INTERFACE I_PersistentEventStorage

METHOD StoreEvent
VAR_INPUT
	stEvent : ST_Event;
END_VAR
END_METHOD

END_INTERFACE

(* stored: Version 1.1.0.1, ProductVersion 3.1.4024.12
   Itf I_PersistentEventStorage: Id {5b8bc0a1-daf5-4b98-9808-63418c12596e}
   Method StoreEvent: Id {f4f5db8c-2cf8-4828-b5c2-b5d4c42af583} *)
